FUNCTION_BLOCK E_D_FF_1 (* Data latch (d) flip flop for 1 BOOL, EO only on change of at least one (generic FB) *)
  (* Standard: 61499-1 Annex A; Description: Copyright (c) 2017, 2026 fortiss GmbH, HR Agrartechnik GmbH This program and the accompanying materials are made available under the terms of the Eclipse Public License 2.0 which is available at https://www.eclipse.org/legal/epl-2.0/ SPDX-License-Identifier: EPL-2.0 *)
  (* Version 1.0, 2026-08-26, Franz Höpfinger, HR Agrartechnik GmbH, E_D_FF extended to 1 BOOL - EO fires only if at least one Di differs from the latched Qi. Service Interface FB, native implementation GEN_E_D_FF (FORTE) required. *)
  PACKAGE iec61499::events;
  {SET_ATTRIBUTE(eclipse4diac::core::GenericClassName, 'GEN_E_D_FF')}
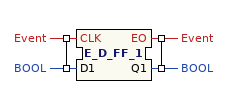
  EVENT_INPUT
    CLK WITH D1; (* Clock *)
  END_EVENT
  EVENT_OUTPUT
    EO WITH Q1; (* Triggered if clock results in a change of at least one Q *)
  END_EVENT
  VAR_INPUT
    D1 : BOOL; (* Value 1 to latch *)
  END_VAR
  VAR_OUTPUT
    Q1 : BOOL; (* Latched value 1 *)
  END_VAR
END_FUNCTION_BLOCK
